// SIMATIC S7-200 project (STEP 7-Micro/WIN), CPU 221 REL 01.10

SYMBOL_TABLE USUARIO1
V1_V2            Q0.0     // Led verde semáforos 1 y 2
A1_A2            Q0.1     // Led amarillo semáforos 1 y 2
R1_R2            Q0.2     // Led rojo semáforos 1 y 2
V3               Q0.3     // Led verde semáforo 3
R3               Q0.4     // Led rojo semáforo 3
V4               Q0.5     // Led verde semáforo 4
A4               Q0.6     // Led amarillo semáforo 4
R4               Q0.7     // Led rojo semáforo 4
V5               Q1.0     // Led verde semáforo 5
R5               Q1.1     // Led rojo semáforo 5
V6               Q1.2     // Led verde semáforo 6
A6               Q1.3     // Led amarillo semáforo 6
R6               Q1.4     // Led rojo semáforo 6
END_SYMBOL_TABLE

ORGANIZATION_BLOCK PRINCIPAL:OB1
TITLE=COMENTARIOS DEL PROGRAMA
BEGIN
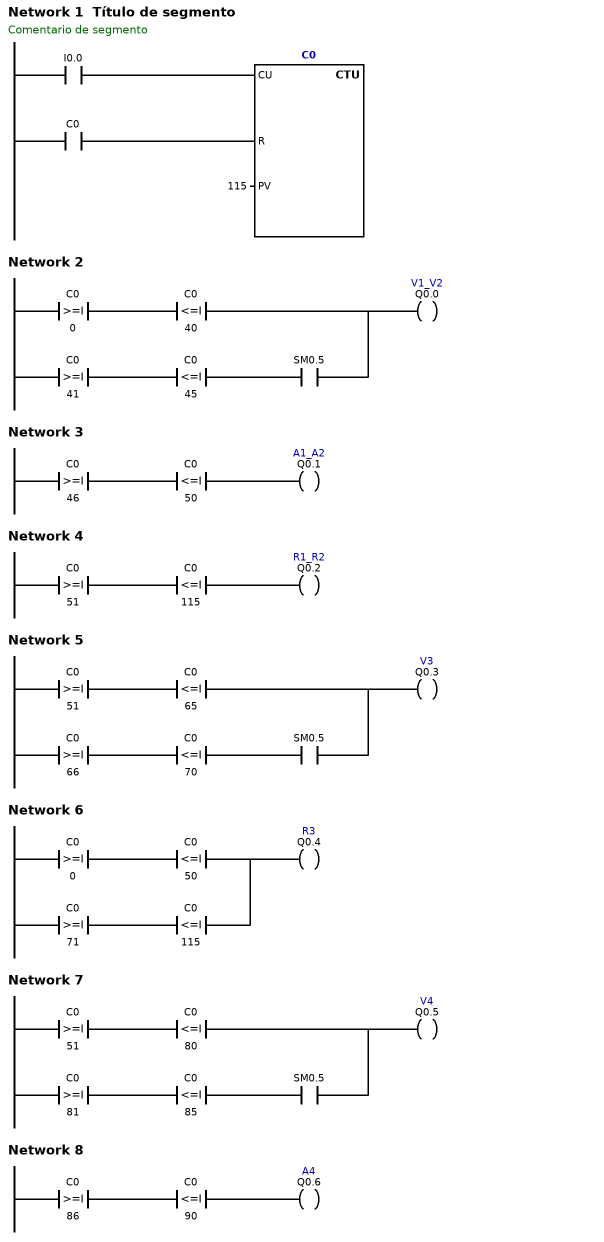
Network 1 // Título de segmento
// Comentario de segmento
LD     I0.0
LD     C0
CTU    C0, 115
Network 2
LDW>=  C0, 0
AW<=   C0, 40
LDW>=  C0, 41
AW<=   C0, 45
A      SM0.5
OLD
=      V1_V2:Q0.0
Network 3
LDW>=  C0, 46
AW<=   C0, 50
=      A1_A2:Q0.1
Network 4
LDW>=  C0, 51
AW<=   C0, 115
=      R1_R2:Q0.2
Network 5
LDW>=  C0, 51
AW<=   C0, 65
LDW>=  C0, 66
AW<=   C0, 70
A      SM0.5
OLD
=      V3:Q0.3
Network 6
LDW>=  C0, 0
AW<=   C0, 50
LDW>=  C0, 71
AW<=   C0, 115
OLD
=      R3:Q0.4
Network 7
LDW>=  C0, 51
AW<=   C0, 80
LDW>=  C0, 81
AW<=   C0, 85
A      SM0.5
OLD
=      V4:Q0.5
Network 8
LDW>=  C0, 86
AW<=   C0, 90
=      A4:Q0.6
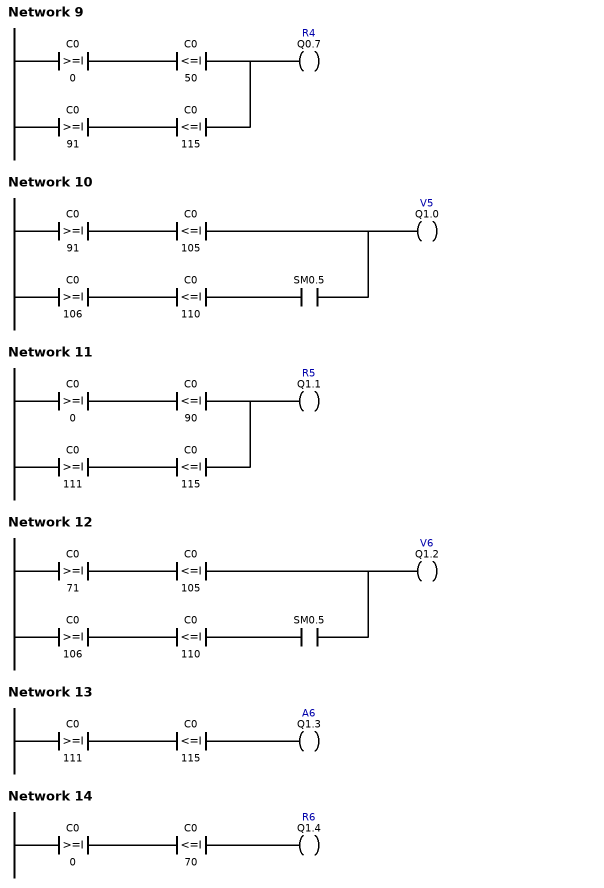
Network 9
LDW>=  C0, 0
AW<=   C0, 50
LDW>=  C0, 91
AW<=   C0, 115
OLD
=      R4:Q0.7
Network 10
LDW>=  C0, 91
AW<=   C0, 105
LDW>=  C0, 106
AW<=   C0, 110
A      SM0.5
OLD
=      V5:Q1.0
Network 11
LDW>=  C0, 0
AW<=   C0, 90
LDW>=  C0, 111
AW<=   C0, 115
OLD
=      R5:Q1.1
Network 12
LDW>=  C0, 71
AW<=   C0, 105
LDW>=  C0, 106
AW<=   C0, 110
A      SM0.5
OLD
=      V6:Q1.2
Network 13
LDW>=  C0, 111
AW<=   C0, 115
=      A6:Q1.3
Network 14
LDW>=  C0, 0
AW<=   C0, 70
=      R6:Q1.4
END_ORGANIZATION_BLOCK
